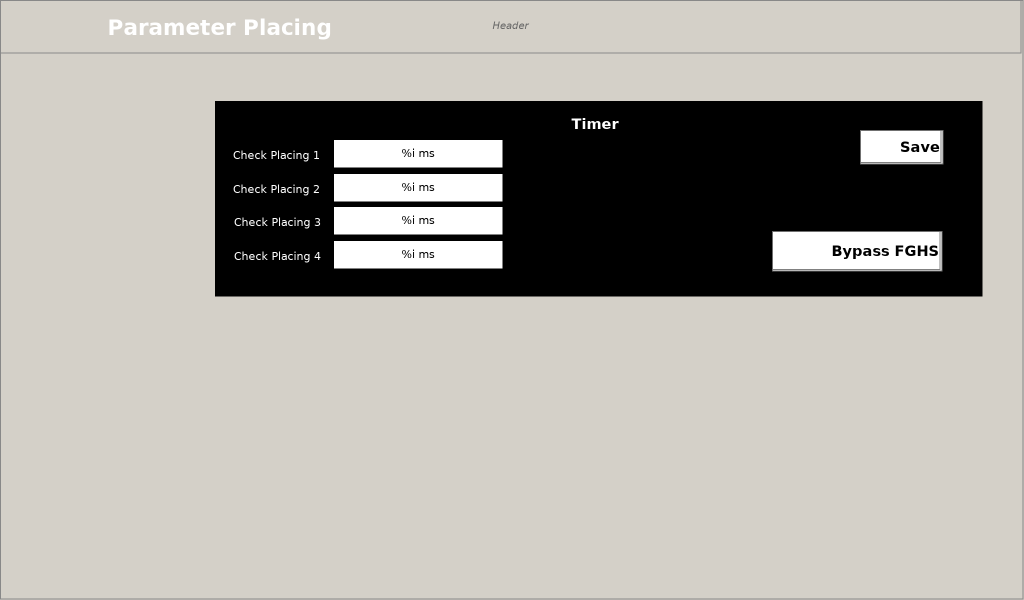
VISUALIZATION MPlacing  // 1024x600
    Frame (0,-2 1021x55)
        shows Header()
    Label (95,15 250x25), "Parameter Placing"
    RoundedRectangle (215,101 767x195)
    Label (243,104 704x40), "Timer"
    Label (230,138 103x35), "Check Placing 1"
    RoundedRectangle (333,139 170x29), "%i ms", text variable: HMI_GVL.Tmr_Placing1
        OnMouseClick: write the text variable via Default
    Button (860,130 83x34), "Save", image: VisuSymbols.Symbols.Save
        tap InputOutput_GVL.TestMode[100]
    Label (230,172 104x35), "Check Placing 2"
    RoundedRectangle (333,173 170x29), "%i ms", text variable: HMI_GVL.Tmr_Placing2
        OnMouseClick: write the text variable via Default
    Label (231,205 102x35), "Check Placing 3"
    RoundedRectangle (333,206 170x29), "%i ms", text variable: HMI_GVL.Tmr_Placing3
        OnMouseClick: write the text variable via Default
    Label (231,239 100x35), "Check Placing 4"
    RoundedRectangle (333,240 170x29), "%i ms", text variable: HMI_GVL.Tmr_Placing4
        OnMouseClick: write the text variable via Default
    Button (772,231 170x40), "Bypass FGHS", colour toggle: HMI_GVL.BypassFGHS, image: VisuSymbols.Symbols.Lock
        toggle HMI_GVL.BypassFGHS
END_VISUALIZATION

(* stored: Version 1.1.0.1, ProductVersion 3.1.4024.12
   Visu MPlacing: Id {9aa48c71-c5e9-4bf3-9649-5a4dc2fa2568} *)
